// TIA Portal V16 export
// export: Created 2022-02-28T20:47:28.5342741Z, ExportSetting WithDefaults, DisplayName Totally Integrated Automation Portal, DisplayVersion V16, DisplayName TIA Portal Version Control Interface, DisplayVersion V16, DisplayName TIA Portal Openness, DisplayVersion V16, DisplayName STEP 7 Professional, DisplayVersion V16, DisplayName STEP 7 Safety, DisplayVersion V16, DisplayName WinCC Advanced, DisplayVersion V16
VAR_GLOBAL   // PLC tag table "01_Entradas"
   MPistilos_Btn_Start AT %I0.0 : Bool;   // Pulsador Start Pistilos
   MPistilos_Btn_Stop AT %I0.1 : Bool;   // Pulsador Stop Pistilos
   MPistilos_Btn_PE AT %I0.2 : Bool;   // Paro Emergencia Pistilos
   MPistilos_Cam_ST AT %I0.3 : Bool;   // Trigger Pistilos Cam 1
   MPentoflex_Btn_Start AT %I0.4 : Bool;   // Pulsador Start Pentoflex
   MPentoflex_Btn_Stop AT %I0.5 : Bool;   // Pulsador Stop Pentonflex
   MPentoflex_Btn_PE AT %I0.6 : Bool;   // Paro Emergencia Pentoflex
   MPentoflex_Cam_ST AT %I0.7 : Bool;   // Trigger Pentoflex Cam 2
END_VAR
